# EPICS substitutions: evrSupport/Db/ioc/bsaBLENEdef.substitutions
#==============================================================================
#
# Abs:  Beam Synchronous Acquisition records for a single
#	bunch length measurement.
#
# Name: bsaBLENEdef.substitutions
#
# Note: Must follow the LCLS naming conventions.
#
#==============================================================================
#
file bsaATTREdef.db
{
#           Device     Attribute       Input            EGU   HOPR  LOPR PREC ADEL  Link
  pattern {   D       , ATTR     ,      I              , EG ,  HO , LO  , PR , AD ,  LNK       , SINK_SIZE}
	  { $(DEVICE) ,$(ATB)RAW ,$(DEVICE):$(ATB)RAW  , "" , 300 , 100 ,  3 , 1  ,  ""       , $(SINK_SIZE\=10) }
	  { $(DEVICE) ,$(ATB)IMAX,$(DEVICE):$(ATB)IMAX , A  , 300 , 100 ,  3 , 1  ,  $(SLCLNK), $(SINK_SIZE\=10) }
}
